(* Schneider Machine Expert - Basic project prg_control, file version 2.7.0.0 *)
(* ProjectInformations: Name=New project *)

HARDWARE
  Cpu 0: TM221M16R/G
  EthernetConfiguration: NetworkName=M221, IpAllocationMode=FixedAddress, IpAddress=0.0.0.0, SubnetMask=0.0.0.0
  SerialLineConfiguration: Baud=Baud19200, Parity=ParityEven, DataBits=DataBits8, StopBits=StopBits1, PhysicalMedium=PhysicalMediumRs485, TransmissionMode=TransmissionModeModbusRtu, SlaveId=1, Addressing=SlaveAddressing
  MastTask: UsePeriodScanMode=false, PeriodScan=100
  FastTask: Period=255
  CpuBehavior: StartingMode=StartAsPreviousState, AutoSaveRamOnEeprom=true, WatchdogPeriod=250

SYMBOLS  (address, symbol, comment, settings)
  %M0       AUX_MOTOR
  %I0.0     I_START  "start process"
  %I0.1     I_STOP  "stop process"
  %I0.5     I_SENSOR  "detecting"
  %Q0.0     Q_MOTOR

POU PRG_Control
  (* SectionNumber=1 *)

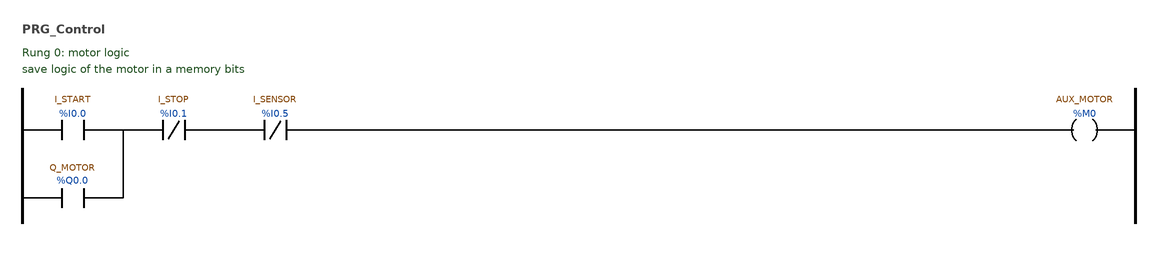

// Rung 0: motor logic
// save logic of the motor in a memory bits
  LD %I0.0                (* I_START *)
  OR %Q0.0                (* Q_MOTOR *)
  ANDN %I0.1              (* I_STOP *)
  ANDN %I0.5              (* I_SENSOR *)
  ST %M0                  (* AUX_MOTOR *)
  // as ST:
  //   AUX_MOTOR := (I_START OR Q_MOTOR) AND NOT I_STOP AND NOT I_SENSOR;

POU PRG OUTPUT
  (* SectionNumber=2 *)

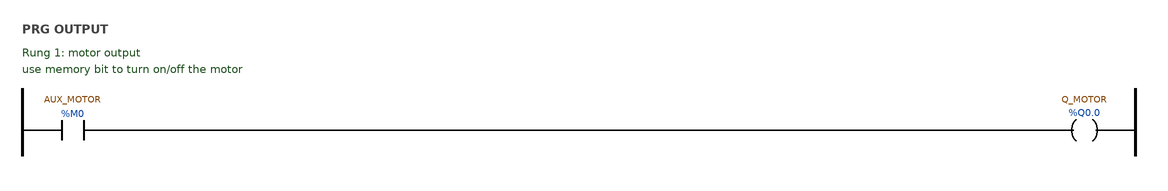

// Rung 1: motor output
// use memory bit to turn on/off the motor
  LD %M0                  (* AUX_MOTOR *)
  ST %Q0.0                (* Q_MOTOR *)
  // as ST:
  //   Q_MOTOR := AUX_MOTOR;
